FUNCTION_BLOCK EL4001
VAR
	_io : EL4xx1_Data;
	{attribute addProperty Name "WcState"}
	_wcState : WcStateBase;
	{attribute addProperty Name "Info data"}
	_infoData : InfoDataAds;
END_VAR

PROPERTY IO : REFERENCE TO EL4xx1_Data
GET
IO REF= _io;
END_GET
END_PROPERTY

PROPERTY WcState : REFERENCE TO WcStateBase
GET
WcState REF= _wcState;
END_GET
END_PROPERTY

END_FUNCTION_BLOCK

(* stored: Version 1.1.0.1, ProductVersion 3.1.4024.9
   POU EL4001: Id {ee5e6bac-f3e2-0b80-2e97-28d5b98745e1}, SpecialFunc None
   Property IO: Id {ed11a8c4-6c91-0b59-1f49-b9fb3b452403}
   Get Get: Id {c74303a0-a253-0cce-1cd3-a89875c0331c}
   Property WcState: Id {06d0258a-0d0b-0a71-1fce-e66fcd353d2c}
   Get Get: Id {3530ce62-9afb-03a2-1117-29fe8e44f4ff} *)
